// TwinCAT 3 PLC project MainPLC
// ProgramVersion: 3.1.4023.0
// libraries:
//   Tc2_MC2, * (Beckhoff Automation GmbH)
//   Tc2_NC, * (Beckhoff Automation GmbH)
//   Tc2_Standard, * (Beckhoff Automation GmbH)
//   Tc2_System, * (Beckhoff Automation GmbH)
//   Tc3_Module, * (Beckhoff Automation GmbH)
//   VisuDialogs, * (System)
// project tree:
//   / GlobalTextList.TcGTLO, PlcTask.TcTTO, Visualization Manager.TcVMO (not stored)
//   POUs/ byteCounter.TcPOU, MAIN.TcPOU, motionChalleng_moveAbs.TcPOU, onOffLed.TcPOU, SevenSegDecoder.TcPOU, sevenSegDecoderV2.TcPOU, sevenSegProg.TcPOU
//   VISUs/ byteCounter.TcVIS, moveAbs.TcVIS, onOffLED.TcVIS, sevenSegmentDisplay.TcVIS
// real-time tasks:
//   TASK PlcTask: cycle T#10ms, priority 20, ADS port 350
// motion (NC):
//   TASK NC-Task 1 SAF: cycle T#2ms, priority 4, ADS port 501
//   TASK NC-Task 1 SVB: cycle T#10ms, priority 8, ADS port 511
//   AXIS Axis 1 (id 1)
// variable links:
//   MainPLC Instance <-> NC-Task 1 SAF/Axes/Axis 1
//     PlcTask Inputs/motionChalleng_moveAbs.myAxis.NcToPlc <-> Outputs/ToPlc
//     PlcTask Outputs/motionChalleng_moveAbs.myAxis.PlcToNc <-> Inputs/FromPlc

CONFIGURATION MainPLC
    RESOURCE PLC ON TwinCAT3
        TASK PlcTask(INTERVAL := T#10ms, PRIORITY := 20);
        PROGRAM MAIN WITH PlcTask : MAIN;
    END_RESOURCE
END_CONFIGURATION

// ---- POUs/MAIN.TcPOU
PROGRAM MAIN
VAR
END_VAR

onOffLed();
byteCounter();
sevenSegProg();
motionChalleng_moveAbs();

END_PROGRAM

// ---- POUs/onOffLed.TcPOU
PROGRAM onOffLed
VAR
    inputSwitch : BOOL;
    outputLED : BOOL;
    rTrig : R_TRIG;
END_VAR

rTrig(CLK:= inputSwitch);

IF rTrig.Q THEN
    outputLED:= NOT outputLED;
END_IF
inputSwitch:= FALSE;

END_PROGRAM

// ---- POUs/byteCounter.TcPOU
PROGRAM byteCounter
VAR
    byteCount : BYTE;
    timer1 : TON;
    timer2 : TON;
    bitRep : ARRAY [0..7] OF BOOL;
    
END_VAR

timer1.IN := TRUE; 
timer1.PT := T#500mS;

IF timer1.Q THEN
    byteCount := byteCount + 1;
    timer1.IN := FALSE;
END_IF

timer1();

bitRep[0] := byteCount.0;
bitRep[1] := byteCount.1;
bitRep[2] := byteCount.2;
bitRep[3] := byteCount.3;
bitRep[4] := byteCount.4;
bitRep[5] := byteCount.5;
bitRep[6] := byteCount.6;
bitRep[7] := byteCount.7;

END_PROGRAM

// ---- POUs/sevenSegProg.TcPOU
PROGRAM sevenSegProg
VAR
digit1Decoder : SevenSegDecoder;
digit2Decoder : SevenSegDecoderV2;
inputDigit : INT := 0;
END_VAR

digit1Decoder(digit:= inputDigit);
digit2Decoder(digit:= inputDigit);

END_PROGRAM

// ---- POUs/SevenSegDecoder.TcPOU
FUNCTION_BLOCK SevenSegDecoder
VAR_INPUT
    digit : INT;
END_VAR
VAR_OUTPUT
    decodedDigit : ARRAY [0..6] OF BOOL;
END_VAR
VAR
    bitA : BOOL;
    bitB : BOOL;
    bitC : BOOL;
    bitD : BOOL;
	inv_bitA: BOOL;
    inv_bitB: BOOL;
    inv_bitC: BOOL;
    inv_bitD: BOOL;
END_VAR

IF digit>9 OR digit<0 THEN
    digit:=0;
END_IF
bitA:= digit.3;
bitB:= digit.2;
bitC:= digit.1;
bitD:= digit.0;
inv_bitA := NOT(bitA);
inv_bitB := NOT(bitB);
inv_bitC := NOT(bitC);
inv_bitD := NOT(bitD);

decodedDigit[0]:= NOT((inv_bitA AND inv_bitB AND inv_bitC AND bitD) OR (bitB AND inv_bitC AND inv_bitD));
decodedDigit[1]:= NOT((bitB AND inv_bitC AND bitD) OR (bitB AND bitC AND inv_bitD));
decodedDigit[2]:= NOT(inv_bitB AND bitC AND inv_bitD);
decodedDigit[3]:= NOT((inv_bitA AND inv_bitB AND inv_bitC AND bitD) OR (bitB AND inv_bitC AND inv_bitD) OR (bitB AND bitC AND bitD));
decodedDigit[4]:= (bitC AND inv_bitD) OR (inv_bitB AND inv_bitD);
decodedDigit[5]:= NOT((inv_bitA AND inv_bitB AND bitD) OR (inv_bitA AND inv_bitB AND bitC) OR (inv_bitA AND bitC AND bitD));
decodedDigit[6]:= NOT((inv_bitA AND inv_bitB AND inv_bitC) OR (bitB AND bitC AND bitD));

END_FUNCTION_BLOCK

// ---- POUs/sevenSegDecoderV2.TcPOU
FUNCTION_BLOCK sevenSegDecoderV2
VAR_INPUT
    digit : INT;
END_VAR
VAR_OUTPUT
    decodedDigit : ARRAY [0..6] OF BOOL;
END_VAR
VAR
    //Lookups
    decoded_0 : ARRAY[0..6] OF BOOL:=[1,1,1,1,1,1,0];
    decoded_1 : ARRAY[0..6] OF BOOL:=[0,1,1,0,0,0,0];
    decoded_2 : ARRAY[0..6] OF BOOL:=[1,1,0,1,1,0,1];
    decoded_3 : ARRAY[0..6] OF BOOL:=[1,1,1,1,0,0,1];
    decoded_4 : ARRAY[0..6] OF BOOL:=[0,1,1,0,0,1,1];
    decoded_5 : ARRAY[0..6] OF BOOL:=[1,0,1,1,0,1,1];
    decoded_6 : ARRAY[0..6] OF BOOL:=[1,0,1,1,1,1,1];
    decoded_7 : ARRAY[0..6] OF BOOL:=[1,1,1,0,0,0,0];
    decoded_8 : ARRAY[0..6] OF BOOL:=[1,1,1,1,1,1,1];
    decoded_9 : ARRAY[0..6] OF BOOL:=[1,1,1,1,0,1,1];
    
END_VAR

IF digit>9 OR digit<0 THEN
    digit:=0;
END_IF

CASE digit OF
    0:
        decodedDigit := decoded_0;
    1:
        decodedDigit := decoded_1;
    2:
        decodedDigit := decoded_2;
    3:
        decodedDigit := decoded_3;
    4:
        decodedDigit := decoded_4;
    5:
        decodedDigit := decoded_5;
    6:
        decodedDigit := decoded_6;
    7:
        decodedDigit := decoded_7;
    8:
        decodedDigit := decoded_8;
    9:
        decodedDigit := decoded_9;                                                                        
END_CASE

END_FUNCTION_BLOCK

// ---- POUs/motionChalleng_moveAbs.TcPOU
PROGRAM motionChalleng_moveAbs
VAR
    myAxis : AXIS_REF;
    mcPower : MC_Power;
    mcMoveAbs : MC_MoveAbsolute;
    highLimitPosition : LREAL := 500;
    lowLimitPosition : LREAL := -5;
    enableAxis : BOOL;
    
    userSetPoint : LREAL;
    defaultVelocity : LREAL := 50;
    executeMoveAbs : BOOL;
END_VAR

mcPower(Axis:= myAxis, Enable_Positive:= highLimit, Enable_Negative:= lowLimit, Enable:= enableAxis);

mcMoveAbs(Axis:= myAxis, Execute:= executeMoveAbs, Position:= userSetPoint, Velocity:= defaultVelocity);
IF mcMoveAbs.Done THEN
    executeMoveAbs:= FALSE;
END_IF

TRANSITION highLimit:
highLimit:= myAxis.NcToPlc.ActPos<highLimitPosition;
END_TRANSITION

TRANSITION lowLimit:
lowLimit:= myAxis.NcToPlc.ActPos>lowLimitPosition;
END_TRANSITION

END_PROGRAM

// ---- GlobalTextList.TcGTLO
TEXTLIST GlobalTextList
  320 = '%.3f'
  37 = '%d'
  441 = '%f.2'
  496 = 'Helpo'
END_TEXTLIST

// ---- VISUs/byteCounter.TcVIS
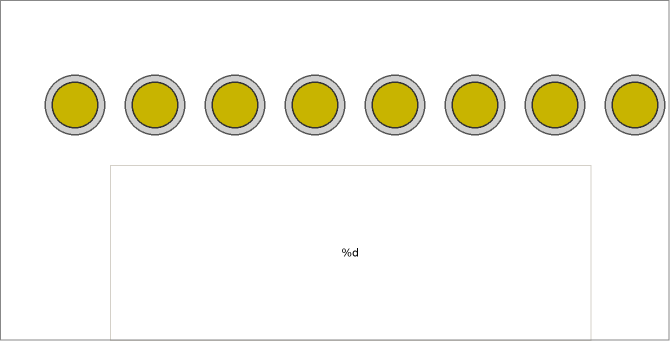
VISUALIZATION byteCounter  // 670x341
    Lamp1 (120,70 70x70), variable: byteCounter.bitRep[6], style: Lamp-Lamp1-Yellow
    Lamp1 (40,70 70x70), variable: byteCounter.bitRep[7], style: Lamp-Lamp1-Yellow
    Lamp1 (280,70 70x70), variable: byteCounter.bitRep[4], style: Lamp-Lamp1-Yellow
    Lamp1 (200,70 70x70), variable: byteCounter.bitRep[5], style: Lamp-Lamp1-Yellow
    Lamp1 (440,70 70x70), variable: byteCounter.bitRep[2], style: Lamp-Lamp1-Yellow
    Lamp1 (360,70 70x70), variable: byteCounter.bitRep[3], style: Lamp-Lamp1-Yellow
    Lamp1 (600,70 70x70), variable: byteCounter.bitRep[0], style: Lamp-Lamp1-Yellow
    Lamp1 (520,70 70x70), variable: byteCounter.bitRep[1], style: Lamp-Lamp1-Yellow
    Textfield (110,165 481x176), "%d", text variable: byteCounter.byteCount
END_VISUALIZATION

// ---- VISUs/moveAbs.TcVIS
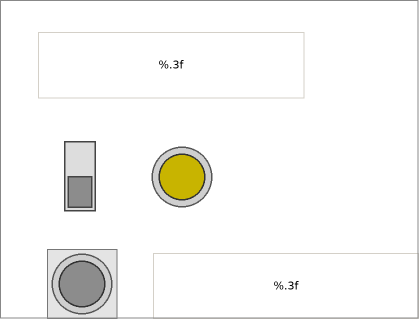
VISUALIZATION moveAbs  // 419x319
    Textfield (38,32 266x66), "%.3f", text variable: motionChalleng_moveAbs.myAxis.NcToPlc.ActPos
    DipSwitch (45,141 70x70), variable: motionChalleng_moveAbs.enableAxis, behaviour: TOGGLE, style: Switch-DipSwitch-Gray
    Lamp1 (147,142 70x70), variable: motionChalleng_moveAbs.mcPower.Status, style: Lamp-Lamp1-Yellow
    PushSwitch (47,249 70x70), variable: motionChalleng_moveAbs.executeMoveAbs, behaviour: TOGGLE, style: Switch-PushSwitch-Gray
    Textfield (153,253 266x66), "%.3f", text variable: motionChalleng_moveAbs.userSetPoint
        OnMouseDown: write motionChalleng_moveAbs.userSetPoint via Default
END_VISUALIZATION

// ---- VISUs/onOffLED.TcVIS
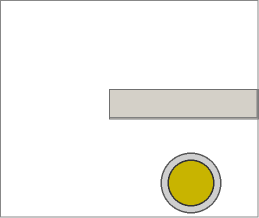
VISUALIZATION onOffLED  // 259x218
    Button (109,89 150x30)
        toggle onOffLed.inputSwitch
    Lamp1 (156,148 70x70), variable: onOffLed.outputLED, style: Lamp-Lamp1-Yellow
END_VISUALIZATION

// ---- VISUs/sevenSegmentDisplay.TcVIS
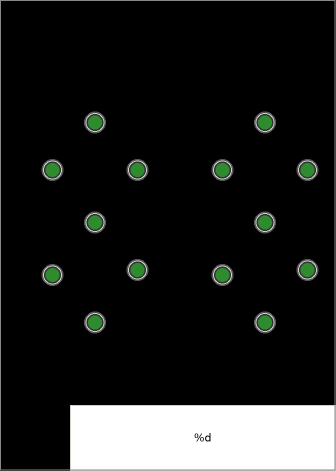
VISUALIZATION sevenSegmentDisplay  // 336x471
    Lamp1 (60,110 70x25), variable: sevenSegProg.digit1Decoder.decodedDigit[0], style: Lamp-Lamp1-Green
    Lamp1 (125,135 25x70), variable: sevenSegProg.digit1Decoder.decodedDigit[1], style: Lamp-Lamp1-Green
    Lamp1 (40,135 25x70), variable: sevenSegProg.digit1Decoder.decodedDigit[5], style: Lamp-Lamp1-Green
    Lamp1 (60,210 70x25), variable: sevenSegProg.digit1Decoder.decodedDigit[6], style: Lamp-Lamp1-Green
    Lamp1 (60,310 70x25), variable: sevenSegProg.digit1Decoder.decodedDigit[3], style: Lamp-Lamp1-Green
    Lamp1 (125,235 25x70), variable: sevenSegProg.digit1Decoder.decodedDigit[2], style: Lamp-Lamp1-Green
    Lamp1 (40,240 25x70), variable: sevenSegProg.digit1Decoder.decodedDigit[4], style: Lamp-Lamp1-Green
    Textfield (70,405 266x66), "%d", text variable: sevenSegProg.inputDigit
        OnMouseClick: write sevenSegProg.inputDigit via Default
    Lamp1 (230,110 70x25), variable: sevenSegProg.digit2Decoder.decodedDigit[0], style: Lamp-Lamp1-Green
    Lamp1 (295,135 25x70), variable: sevenSegProg.digit2Decoder.decodedDigit[1], style: Lamp-Lamp1-Green
    Lamp1 (210,135 25x70), variable: sevenSegProg.digit2Decoder.decodedDigit[5], style: Lamp-Lamp1-Green
    Lamp1 (230,210 70x25), variable: sevenSegProg.digit2Decoder.decodedDigit[6], style: Lamp-Lamp1-Green
    Lamp1 (230,310 70x25), variable: sevenSegProg.digit2Decoder.decodedDigit[3], style: Lamp-Lamp1-Green
    Lamp1 (295,235 25x70), variable: sevenSegProg.digit2Decoder.decodedDigit[2], style: Lamp-Lamp1-Green
    Lamp1 (210,240 25x70), variable: sevenSegProg.digit2Decoder.decodedDigit[4], style: Lamp-Lamp1-Green
END_VISUALIZATION
